{attribute 'qualified_only'}
{attribute 'strict'}
TYPE STATI :
(
	S0 := 0, S1, S2, S3, SE, SA
);
END_TYPE

(* stored: Version 1.1.0.1, ProductVersion 3.1.4024.12
   EnumerationTextList DUT: Id {de053a43-a5fe-45fc-9c72-dc62d4688ffa} *)
